// TwinCAT 3 PLC project Contol
// ProgramVersion: 3.1.4023.0
// libraries:
//   Tc2_MC2, * (Beckhoff Automation GmbH)
//   Tc2_MC2_Camming, * (Beckhoff Automation GmbH)
//   Tc2_Standard, * (Beckhoff Automation GmbH)
//   Tc2_System, * (Beckhoff Automation GmbH)
//   Tc2_Utilities, * (Beckhoff Automation GmbH)
//   Tc3_Module, * (Beckhoff Automation GmbH)
//   VisuSymbols,3.5.10.0,System
// project tree:
//   / GlobalTextList.TcGTLO, PlcTask.TcTTO, Visualization Manager.TcVMO (not stored)
//   GVLs/ GVL_UserParamerts.TcGVL
//   POUs/ FB_CsvRead_CamTable.TcPOU, MAIN.TcPOU
//   VISUs/ Visualization.TcVIS
// real-time tasks:
//   TASK PlcTask: cycle T#10ms, priority 20, ADS port 350
// motion (NC):
//   TASK NC-Task 1 SAF: cycle T#2ms, priority 4, ADS port 501
//   TASK NC-Task 1 SVB: cycle T#10ms, priority 8, ADS port 511
//   AXIS master (id 1)
//     OtherSettings: AllowMotionCmdToSlave=true
//     encoder EncType=1
//     drive DrvType=5
//       Analog: TorqueSetpointScale=10, ScaleFactorActTorque=0.1
//       TimeComp: TaskDelayCycles=1
//     controller CtrType=1
//       CtrPara: PriorControlFactor=1
//         Observer: BandWidth=20
//   AXIS Axis 1 (id 2)
//     OtherSettings: AllowMotionCmdToSlave=true
//     encoder EncType=1
//     drive DrvType=5
//       Analog: TorqueSetpointScale=10, ScaleFactorActTorque=0.1
//       TimeComp: TaskDelayCycles=1
//     controller CtrType=1
//       CtrPara: PriorControlFactor=1
//         Observer: BandWidth=20
//   AXIS Axis 2 (id 3)
//     OtherSettings: AllowMotionCmdToSlave=true
//     encoder EncType=1
//     drive DrvType=5
//       Analog: TorqueSetpointScale=10, ScaleFactorActTorque=0.1
//       TimeComp: TaskDelayCycles=1
//     controller CtrType=1
//       CtrPara: PriorControlFactor=1
//         Observer: BandWidth=20
//   AXIS Axis 3 (id 4)
//     OtherSettings: AllowMotionCmdToSlave=true
//     encoder EncType=1
//     drive DrvType=5
//       Analog: TorqueSetpointScale=10, ScaleFactorActTorque=0.1
//       TimeComp: TaskDelayCycles=1
//     controller CtrType=1
//       CtrPara: PriorControlFactor=1
//         Observer: BandWidth=20
//   AXIS Axis 4 (id 5)
//     OtherSettings: AllowMotionCmdToSlave=true
//     encoder EncType=1
//     drive DrvType=5
//       Analog: TorqueSetpointScale=10, ScaleFactorActTorque=0.1
//       TimeComp: TaskDelayCycles=1
//     controller CtrType=1
//       CtrPara: PriorControlFactor=1
//         Observer: BandWidth=20
//   AXIS Axis 5 (id 6)
//     OtherSettings: AllowMotionCmdToSlave=true
//     encoder EncType=1
//     drive DrvType=5
//       Analog: TorqueSetpointScale=10, ScaleFactorActTorque=0.1
//       TimeComp: TaskDelayCycles=1
//     controller CtrType=1
//       CtrPara: PriorControlFactor=1
//         Observer: BandWidth=20
// variable links:
//   Contol/Contol Instance <-> NC-Task 1 SAF/Axes/Axis 1
//     PlcTask Inputs/MAIN.AxMotor[0].NcToPlc <-> Outputs/ToPlc
//     PlcTask Outputs/MAIN.AxMotor[0].PlcToNc <-> Inputs/FromPlc
//   Contol/Contol Instance <-> NC-Task 1 SAF/Axes/Axis 2
//     PlcTask Inputs/MAIN.AxMotor[1].NcToPlc <-> Outputs/ToPlc
//     PlcTask Outputs/MAIN.AxMotor[1].PlcToNc <-> Inputs/FromPlc
//   Contol/Contol Instance <-> NC-Task 1 SAF/Axes/Axis 3
//     PlcTask Inputs/MAIN.AxMotor[2].NcToPlc <-> Outputs/ToPlc
//     PlcTask Outputs/MAIN.AxMotor[2].PlcToNc <-> Inputs/FromPlc
//   Contol/Contol Instance <-> NC-Task 1 SAF/Axes/Axis 4
//     PlcTask Inputs/MAIN.AxMotor[3].NcToPlc <-> Outputs/ToPlc
//     PlcTask Outputs/MAIN.AxMotor[3].PlcToNc <-> Inputs/FromPlc
//   Contol/Contol Instance <-> NC-Task 1 SAF/Axes/Axis 5
//     PlcTask Inputs/MAIN.AxMotor[4].NcToPlc <-> Outputs/ToPlc
//     PlcTask Outputs/MAIN.AxMotor[4].PlcToNc <-> Inputs/FromPlc
//   Contol/Contol Instance <-> NC-Task 1 SAF/Axes/master
//     PlcTask Inputs/MAIN.AXMaster.NcToPlc <-> Outputs/ToPlc
//     PlcTask Outputs/MAIN.AXMaster.PlcToNc <-> Inputs/FromPlc

CONFIGURATION Contol
    RESOURCE PLC ON TwinCAT3
        TASK PlcTask(INTERVAL := T#10ms, PRIORITY := 20);
        PROGRAM MAIN WITH PlcTask : MAIN;
    END_RESOURCE
END_CONFIGURATION

// ---- GVLs/GVL_UserParamerts.TcGVL
//{attribute 'qualified_only'}
VAR_GLOBAL CONSTANT
	// kinetic parameters
	lrVelocity						: REAL		:= 1000;
	lrAcceleration					: REAL		:= 1000;
	lrDeceleration					: REAL		:= 1000;
	
	// show parameters
	rShowVelocity					: REAL		:= 100;
	rShowAcceleration				: REAL		:= 1000;
	rShowDeceleration				: REAL		:= 1000;
	
	// csv file parameters
	iMaxPoints						: INT		:= 5864;		// Maximum number of frames/rows/required positions 32.000 -> Activate Configuration
	iMotorsNum						: INT		:= 5;			// Fixed
	sFileDir						: STRING	:= 'C:\Users\Amr Awad\Desktop\TC_AxesSimulator\_ShowFiles_\';
	sFileName						: STRING	:= 'gesamt_show.csv';
END_VAR
VAR_GLOBAL PERSISTENT
	aa2lrTable						: ARRAY[0..iMotorsNum-1] OF ARRAY[0..iMaxPoints-1,0..1] OF LREAL;
END_VAR

// ---- POUs/MAIN.TcPOU
PROGRAM MAIN
VAR
	fbTimeout						: TON;
	
	(* GUI Parameters *)
	// User Control
	boShowLoad						: BOOL;
	boShowStart						: BOOL;
	boShowPause						: BOOL;
	boShowStop						: BOOL;
	
	(* Show Functions & Parameters *)
	// 1. csv file loading
	fbCsvRead						: FB_CsvRead_CamTable;
	iFrames							: INT;
	boShowLoadError					: BOOL;
	boShowLoading					: BOOL;
	boShowLoaded					: BOOL;
	i								: INT;
	iTable							: INT	:= 0;
	
	// 2. show manupulation
	iShowState						: INT := 0;
	
	// camming table
	TableCamRef						: ARRAY[0..iMotorsNum-1] OF MC_CAM_REF;
	MC_CamTableSelect				: MC_CamTableSelect;
	MC_ReadCamTableCharacteristics	: ARRAY[0..iMotorsNum-1] OF MC_ReadCamTableCharacteristics;
	MC_TableCharacValues			: ARRAY[0..iMotorsNum-1] OF MC_TableCharacValues;
	
	// 1. Master Axis
	AXMaster						: AXIS_REF;
	fbMasterEnable					: MC_Power;
	fbMasterSetPosition				: MC_SetPosition;
	fbMasterMoveAbs					: MC_MoveAbsolute;
	fbMasterStop					: MC_Stop;
	fbMasterReset					: MC_Reset;
	
	boMasterEnable					: BOOL;
	boMasterSetPosition				: BOOL;
	boMasterMovAbs					: BOOL;
	rMasterTargetPosition			: REAL;
	boMasterStop					: BOOL;
	boShowPauseLatch				: BOOL;
	boShowStopLatch					: BOOL;
	boMasterReset					: BOOL;
	
	// 2. Slave Axes
	AxMotor							: ARRAY[0..iMotorsNum-1] OF AXIS_REF;
	fbEnable						: ARRAY[0..iMotorsNum-1] OF MC_Power;
	fbMoveAbs						: ARRAY[0..iMotorsNum-1] OF MC_MoveAbsolute;
	ST_CamInOptions					: ST_CamInOptions;	// Data Type deceleration — MC_CamIn input
	fbCamIn							: ARRAY[0..iMotorsNum-1] OF MC_CamIn;
	fbCamOut						: ARRAY[0..iMotorsNum-1] OF MC_CamOut;
	fbReset							: ARRAY[0..iMotorsNum-1] OF MC_Reset;
	
	boEnable						: BOOL;
	boEnabled						: BOOL;
	boMoveAbs						: BOOL;
	boMoveAbsDone					: BOOL;
	boMoveAbsError					: BOOL;
	boAxCamIn						: BOOL	:= FALSE;
	boAxCamInDone					: BOOL;
	boAxCamOut						: BOOL	:= FALSE;
	boAxCamOutDone					: BOOL;
	boReset							: BOOL;
	
	boShowActived					: BOOL;
END_VAR

// General
boShowLoading										:= fbCsvRead.OUT_boBusy;
boShowLoaded										:= aa2lrTable[iMotorsNum-1][iMaxPoints-1,0] <> 0 AND NOT fbCsvRead.OUT_boBusy;

fbTimeout();

// Logic Control
IF NOT boShowActived THEN
	fbCsvRead(
		IN_smaxDirectoryName		 				:= sFileDir, 
		IN_sFileName								:= sFileName, 
		IN_sColumnSeparator							:= ',', 
		IN_iMotorsNr								:= iMotorsNum, 
		IN_boStartReading							:= boShowLoad, 
		IN_paa2lrTable								:= ADR(aa2lrTable), 
		OUT_boError									=> boShowLoadError);
	IF fbCsvRead.OUT_boDone AND NOT fbCsvRead.OUT_boError THEN
		iFrames										:= fbCsvRead.OUT_iRowsnNumber;
		boShowLoad									:= FALSE;
	ELSIF fbCsvRead.OUT_boDone AND fbCsvRead.OUT_boError THEN
		boShowLoad									:= FALSE;
	END_IF
	IF boShowLoaded AND boShowStart THEN
		boShowActived								:= TRUE;
		iShowState									:= 10;
	END_IF
ELSE
	CASE iShowState OF
		0:		// Idle
			boShowActived							:= FALSE;
			boShowPauseLatch						:= FALSE;
			boShowStopLatch							:= FALSE;
			
		10:		// preparing camming referencing
			rMasterTargetPosition					:= LREAL_TO_REAL(aa2lrTable[0][iMaxPoints-1,0]);	// last time stamp in the table
			FOR i := 0 TO iMotorsNum - 1 DO
				TableCamRef[i].pArray				:= ADR(aa2lrTable[i]);
				TableCamRef[i].ArraySize			:= SIZEOF(aa2lrTable[i]);
				TableCamRef[i].TableType			:= MC_TABLETYPE_NONEQUIDISTANT;
				TableCamRef[i].NoOfRows				:= INT_TO_UDINT(iMaxPoints);
				TableCamRef[i].NoOfColumns			:= 2;
			END_FOR
			iShowState								:= 20;
			
		20:		// select camming table
			MC_CamTableSelect(
				Master								:= AxMaster, 
				Slave								:= AxMotor[iTable], 
				CamTable							:= TableCamRef[iTable], 
				Execute								:= TRUE, 
				Periodic							:= FALSE, 
				MasterAbsolute						:= TRUE, 
				SlaveAbsolute						:= TRUE, 
				CamTableID							:= INT_TO_UDINT(iTable+1), 
				Done=> , 
				Busy=> , 
				Error=> , 
				ErrorID=> );
			IF MC_CamTableSelect.Done AND NOT MC_CamTableSelect.Error THEN
				iTable								:= iTable + 1;
				MC_CamTableSelect(	
					Master							:= AxMaster, 
					Slave							:= AxMotor[iTable], 
					CamTable						:= TableCamRef[iTable],
					Execute							:= FALSE);
				IF iTable = iMotorsNum-1 THEN
					iTable							:= 0;
					iShowState						:= 30;
				ELSE
					//
				END_IF
			ELSIF MC_CamTableSelect.Error THEN
				MC_CamTableSelect(	
					Master							:= AxMaster, 
					Slave							:= AxMotor[iTable], 
					CamTable						:= TableCamRef[iTable],
					Execute							:= FALSE);
				iTable								:= 0;
			END_IF
			
		30:		// kinetic initialization
			fbTimeout.IN							:= TRUE;
			fbTimeout.PT							:= T#5S;
			boMasterEnable							:= TRUE;
			boEnable								:= TRUE;
			boEnabled								:= AXMaster.NcToPlc.StateDWord.0;
			FOR i := 0 TO iMotorsNum - 1 DO
				boEnabled							:= boEnabled AND AxMotor[i].NcToPlc.StateDWord.0;
			END_FOR
			IF boEnabled THEN
				fbTimeout.IN						:= FALSE;
				iShowState							:= 40;
			ELSIF fbTimeout.Q THEN
				fbTimeout.IN						:= FALSE;
				// Error
			END_IF
			
		40:		// Master position reset
			boMasterSetPosition						:= TRUE;
			IF fbMasterSetPosition.Done THEN
				boMasterSetPosition					:= FALSE;
				iShowState							:= 50;
			ELSIF fbMasterSetPosition.Error THEN
				boMasterSetPosition					:= FALSE;
				// Error
			END_IF
			
		50:		// move all axes to the home position
			fbTimeout.IN							:= TRUE;
			fbTimeout.PT							:= T#5S;
			boMoveAbs								:= TRUE;
			boMoveAbsDone							:= TRUE;
			boMoveAbsError							:= FALSE;
			FOR i := 0 TO iMotorsNum - 1 DO
				boMoveAbsDone						:= boMoveAbsDone AND fbMoveAbs[i].Done;
				boMoveAbsError						:= boMoveAbsError OR fbMoveAbs[i].Error;
			END_FOR
			IF boMoveAbsDone AND NOT boMoveAbsError THEN
				fbTimeout.IN						:= FALSE;
				boMoveAbs							:= FALSE;
				iShowState							:= 60;
			ELSIF boMoveAbsError THEN
				fbTimeout.IN						:= FALSE;
				boMoveAbs							:= FALSE;
				// Error
			ELSIF fbTimeout.Q THEN
				fbTimeout.IN						:= FALSE;
				// Error
			END_IF
			
		60:		// couple axes
			fbTimeout.IN							:= TRUE;
			fbTimeout.PT							:= T#5S;
			boAxCamIn								:= TRUE;
			boAxCamInDone							:= TRUE;
			FOR i := 0 TO iMotorsNum - 1 DO
				boAxCamInDone						:= boAxCamInDone AND fbCamIn[i].InSync AND NOT fbCamIn[i].Error;
				IF fbCamIn[i].Error THEN
					// Error
				END_IF
			END_FOR
			IF boAxCamInDone THEN
				fbTimeout.IN						:= FALSE;
				boAxCamIn							:= FALSE;
				iShowState							:= 70;
			ELSIF fbTimeout.Q THEN
				fbTimeout.IN						:= FALSE;
				// Error
			END_IF
			
		70:		// move master axis
			boMasterMovAbs							:= TRUE;
			IF fbMasterMoveAbs.Busy THEN
				boMasterMovAbs						:= FALSE;
				iShowState							:= 75;
			END_IF
			
		75:		// check show end
			IF fbMasterMoveAbs.Done THEN
				iShowState							:= 80;
			END_IF
			IF boShowPause THEN
				boMasterStop						:= TRUE;
				boShowPauseLatch					:= TRUE;
				iShowState							:= 77;
			ELSIF boShowStop THEN
				boMasterStop						:= TRUE;
				boShowStopLatch						:= TRUE;
				iShowState							:= 77;
			END_IF
			
		77:		// stop check
			boMasterStop							:= FALSE;
			IF fbMasterStop.Done THEN
				iShowState							:= 78;
			END_IF
			
		78:		// decision making
			IF boShowPauseLatch AND boShowStart THEN
				boShowPauseLatch					:= FALSE;
				iShowState							:= 70;
			END_IF
			IF boShowStopLatch THEN
				iShowState							:= 80;
			END_IF
			
		80:		// decouple axes
			fbTimeout.IN							:= TRUE;
			fbTimeout.PT							:= T#5S;
			boAxCamOut								:= TRUE;
			boAxCamOutDone							:= TRUE;
			FOR i := 0 TO iMotorsNum - 1 DO
				boAxCamOutDone						:= boAxCamOutDone AND fbCamOut[i].Done AND NOT fbCamOut[i].Error;
				IF fbCamOut[i].Error THEN
					// Error
				END_IF
			END_FOR
			IF boAxCamOutDone THEN
				fbTimeout.IN						:= FALSE;
				boAxCamOut							:= FAlse;
				IF boShowStopLatch THEN
					boShowStopLatch					:= FALSE;
					iShowState						:= 0;
				ELSE
					iShowState						:= 40;
				END_IF
			ELSIF fbTimeout.Q THEN
				fbTimeout.IN						:= FALSE;
				// Error
			END_IF
	END_CASE
END_IF

(* Cyclic Calls *)
// 1. Master Axis
fbMasterEnable(
	Axis											:= AxMaster, 
	Enable											:= boMasterEnable, 
	Enable_Positive									:= TRUE, 
	Enable_Negative									:= TRUE, 
	Override										:= 100, 
	BufferMode										:= MC_Aborting, 
	Options:= , 
	Status=> , 
	Busy=> , 
	Active=> , 
	Error=> , 
	ErrorID=> );

fbMasterSetPosition(
	Axis											:= AxMaster, 
	Execute											:= boMasterSetPosition, 
	Position										:= 0, 
	Mode:= , 
	Options:= , 
	Done=> , 
	Busy=> , 
	Error=> , 
	ErrorID=> );

fbMasterMoveAbs(
	Axis											:= AxMaster, 
	Execute											:= boMasterMovAbs, 
	Position										:= rMasterTargetPosition, 
	Velocity										:= rShowVelocity, 
	Acceleration									:= rShowAcceleration, 
	Deceleration									:= rShowDeceleration, 
	Jerk:= , 
	BufferMode:= , 
	Options:= , 
	Done=> , 
	Busy=> , 
	Active=> , 
	CommandAborted=> , 
	Error=> , 
	ErrorID=> );

fbMasterStop(
	Axis											:= AxMaster, 
	Execute											:= boMasterStop, 
	Deceleration:= , 
	Jerk:= , 
	Options:= , 
	Done=> , 
	Busy=> , 
	Active=> , 
	CommandAborted=> , 
	Error=> , 
	ErrorID=> );

fbMasterReset(
	Axis											:= AxMaster, 
	Execute											:= boMasterReset, 
	Done=> , 
	Busy=> , 
	Error=> , 
	ErrorID=> );

// 2. Pendulum Axis
FOR i := 0 TO iMotorsNum-1 DO
	fbEnable[i](
		Axis										:= AxMotor[i], 
		Enable										:= boEnable, 
		Enable_Positive								:= TRUE, 
		Enable_Negative								:= TRUE, 
		Override:= , 
		BufferMode:= , 
		Options:= , 
		Status=> , 
		Busy=> , 
		Active=> , 
		Error=> , 
		ErrorID=> );
	
	fbMoveAbs[i](
		Axis										:= AxMotor[i], 
		Execute										:= boMoveAbs, 
		Position									:= aa2lrTable[i][0, 1], 
		Velocity									:= lrVelocity, 
		Acceleration								:= lrAcceleration, 
		Deceleration								:= lrDeceleration, 
		Jerk:= , 
		BufferMode:= , 
		Options:= , 
		Done=> , 
		Busy=> , 
		Active=> , 
		CommandAborted=> , 
		Error=> , 
		ErrorID=> );
	
	fbCamIn[i](
		Master										:= AxMaster, 
		Slave										:= AxMotor[i], 
		Execute										:= boAxCamIn, 
		MasterOffset								:= 0, 
		SlaveOffset									:= 0, 
		MasterScaling								:= 1, 
		SlaveScaling								:= 1, 
		StartMode:= , 
		CamTableID									:= 1, 
		BufferMode:= , 
		Options										:= ST_CamInOptions, 
		//InterpolationType							:= MC_InterpolationType_Spline, 
		InSync=> , 
		Busy=> , 
		Active=> , 
		CommandAborted=> , 
		Error=> , 
		ErrorID=> );
	
	fbCamOut[i](
		Slave										:= AxMotor[i], 
		Execute										:= boAxCamOut, 
		Options:= , 
		Done=> , 
		Busy=> , 
		Error=> , 
		ErrorID=> );
	
	fbReset[i](
		Axis										:= AxMotor[i], 
		Execute										:= boReset, 
		Done=> , 
		Busy=> , 
		Error=> , 
		ErrorID=> );
END_FOR

END_PROGRAM

// ---- POUs/FB_CsvRead_CamTable.TcPOU
FUNCTION_BLOCK FB_CsvRead_CamTable
VAR_INPUT
	IN_smaxDirectoryName				: T_MaxString;
	IN_sFileName						: STRING;
	IN_sColumnSeparator					: STRING;
	IN_iMotorsNr						: INT;
	IN_boStartReading					: BOOL;
	IN_paa2lrTable						: POINTER TO ARRAY[0..iMotorsNum-1] OF ARRAY[0..iMaxPoints-1,0..1] OF LREAL;
END_VAR
VAR_OUTPUT
	OUT_boBusy							: BOOL;		// Reading active
	OUT_boDone							: BOOL;		// Reading Done user-defined flag
	OUT_boError							: BOOL;
	OUT_iReadingError					: INT;		// Reading error user-defined flag; 0:Clear, 1:Opening, 2:Getting
	OUT_iRowsnNumber					: INT;		// Number of actual read rows
	//OUT_arTableColumn					: ARRAY[0..iMotorsNum] OF ARRAY[0..iMaxPoints-1] OF REAL;
END_VAR

VAR
	ReadCSV								: R_TRIG;
	iStep								: INT;						// identifier of the execution sequence — State index
	
	fbFileOpen							: FB_FileOpen;				// Opens file
	fbFileGets							: FB_FileGets;				// Reads text data from the opened file
	fbReader							: FB_CSVMemBufferReader;	// Helper function block used to parse CSV data bytes
	fbFileClose							: FB_FileClose;				// Closes file
	
	sPathName							: T_MaxString;
	nMode								: DWORD := FOPEN_MODEREAD OR FOPEN_MODEBINARY;	(* FileOpen input *)
	bBusy								: BOOL;											(* Internal Busy flag *)
	nErrId								: UDINT;										(* Block output *)
	hFile								: UINT	:= 0;									(* File handle of the source file *)
	
	iRow								: INT;											// Row number (record)
	iColumn								: INT;											// Column number (record field)
	
	lrDummy								: LREAL;
END_VAR

ReadCSV(CLK								:= IN_boStartReading);	// Latching the start reading command
OUT_boBusy								:= iStep <> 0;			// Busy as long as state machine running

// Column Separator selection
IF IN_sColumnSeparator = ',' THEN
	DEFAULT_CSV_FIELD_SEP				:= 16#2C;				// American Separator (,) 16#2C
ELSIF IN_sColumnSeparator = ';' THEN
	DEFAULT_CSV_FIELD_SEP				:= 16#3B;				// European Separator (;) 16#3B
END_IF

CASE iStep OF 
	0:		// Sleep Mode — wait till the starting signal is triggered
		sPathName						:= CONCAT(IN_smaxDirectoryName, IN_sFileName);
		fbFileOpen(bExecute				:= FALSE);
		fbFileGets(bExecute				:= FALSE);
		IF ReadCSV.Q THEN	// Reset parameters — Transition to the next step
			OUT_boDone			:= FALSE;
			OUT_iReadingError			:= 0;
			MEMSET(IN_paa2lrTable, 0, SIZEOF(IN_paa2lrTable^));
			bBusy						:= TRUE;
			OUT_boError					:= FALSE;
			nErrId						:= 0;
			hFile						:= 0;
			iRow						:= 0;
			iStep						:= 10;
		END_IF
	
	10:		// File Opening Command
		fbFileOpen(	
			sPathName					:= sPathName, 
			nMode						:= nMode, 
			bExecute					:= TRUE, 
			bError						=> OUT_boError, 
			nErrID 						=> nErrID, 
			hFile						=> hFile );
		IF NOT fbFileOpen.bBusy THEN
			IF NOT fbFileOpen.bError THEN
				fbFileOpen(bExecute		:= FALSE);
				iStep					:= 20;      // File opened & without error
			ELSE
				fbFileOpen(bExecute		:= FALSE);
				iStep					:= 100;    // Error — File not found!
				OUT_iReadingError		:= 1;
			END_IF
		END_IF
		
	20:		// Data Getting Command
		fbFileGets(	
			hFile						:= hFile, 
			bExecute					:= TRUE, 
			bError						=> OUT_boError);
		IF NOT fbFileGets.bBusy THEN
			IF NOT fbFileGets.bError THEN
				IF fbFileGets.bEOF THEN
					fbFileGets(bExecute	:= FALSE);
					iStep				:= 40;		// .csv file end is reached — Close File
				ELSE
					fbFileGets(bExecute	:= FALSE);
					iStep				:= 30;		// Parse text data
				END_IF
			ELSE
				iStep					:= 100;		// Error — During the excution!
				OUT_iReadingError		:= 2;
			END_IF		
		END_IF
		
	30:		// Parse text data
		fbReader(	
			eCmd						:= eEnumCmd_First, 
			pBuffer						:= ADR(fbFileGets.sLine), 
			cbBuffer					:= SIZEOF(fbFileGets.sLine));	// Read first field value — given from the manual
		IF fbReader.bOk THEN
			lrDummy						:= STRING_TO_LREAL(fbReader.getValue);
			FOR iColumn := 0 TO IN_iMotorsNr-1 DO
				fbReader(	
					eCmd				:= eEnumCmd_Next, 
					pBuffer				:= ADR(fbFileGets.sLine), 
					cbBuffer			:= SIZEOF(fbFileGets.sLine));
				IN_paa2lrTable^[iColumn][iRow,0]	:= lrDummy;								// Master Axis Positions
				IN_paa2lrTable^[iColumn][iRow,1]	:= STRING_TO_REAL(fbReader.getValue);	// Motors Axes Positions
			END_FOR
			iRow						:= iRow +1;		// Increment number of read records
			iStep						:= 20;			// Read new row
		END_IF
	
	40:		// Close source file command
		OUT_iRowsnNumber				:= iRow;
		fbFileClose(	
			hFile						:= hFile, 
			bExecute					:= TRUE, 
			bError						=> OUT_boError);
		IF NOT fbFileClose.bBusy THEN
			fbFileClose(bExecute		:= FALSE);
			hFile						:= 0;
			iStep						:= 100;
		END_IF
	
	100:	// Error OR ready step => cleanup
		IF ( hFile <> 0 ) THEN
			iStep						:= 10;		// Close the source file and cleanup hFile
		ELSE
			bBusy						:= FALSE;	// Lowering the Busy flag
			OUT_boDone			:= TRUE;	// Ending Service Routine flag
			iStep						:= 0;		// Ready for a new run when triggered/called
		END_IF
END_CASE

END_FUNCTION_BLOCK

// ---- GlobalTextList.TcGTLO
TEXTLIST GlobalTextList
  628 = 'Axes Coupled'
  409 = 'Control'
  464 = 'Feadback'
  166 = 'Show Activated'
  915 = 'Show Load'
  700 = 'Show Loaded'
  942 = 'Show Loading'
  86 = 'Show Pause'
  299 = 'Show Running'
  447 = 'Show Start'
  735 = 'Show Stop'
END_TEXTLIST

// ---- VISUs/Visualization.TcVIS
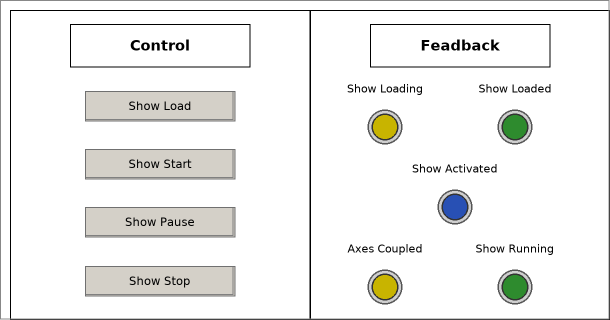
VISUALIZATION Visualization  // 610x320
    Rectangle (310,10 300x310)
    Rectangle (10,10 300x310)
    Button (85,91 150x30), "Show Load", input disabled if: MAIN.boShowActived OR MAIN.fbCsvRead.OUT_boBusy
        tap MAIN.boShowLoad
    Rectangle (70,24 180x43), "Control"
    Button (85,149 150x30), "Show Start", input disabled if: (MAIN.boShowActived AND NOT MAIN.boShowPauseLatch)OR MAIN.fbCsvRead.OUT_boBusy
        tap MAIN.boShowStart
    Button (85,207 150x30), "Show Pause", input disabled if: NOT MAIN.fbMasterMoveAbs.Busy
        tap MAIN.boShowPause
    Button (85,266 150x30), "Show Stop", input disabled if: NOT MAIN.fbMasterMoveAbs.Busy
        tap MAIN.boShowStop
    Rectangle (370,24 180x43), "Feadback"
    Lamp1 (365,107 40x40), variable: MAIN.boShowLoading, style: Lamp-Lamp1-Yellow
    Rectangle (335,79 100x20), "Show Loading"
    Lamp1 (495,107 40x40), variable: MAIN.boShowLoaded, style: Lamp-Lamp1-Green
    Rectangle (465,79 100x20), "Show Loaded"
    Lamp1 (435,187 40x40), variable: MAIN.boShowActived, style: Lamp-Lamp1-Blue
    Rectangle (405,159 100x20), "Show Activated"
    Lamp1 (365,267 40x40), variable: MAIN.AXMaster.NcToPlc.CoupleState = 1, style: Lamp-Lamp1-Yellow
    Rectangle (335,239 100x20), "Axes Coupled"
    Lamp1 (495,267 40x40), variable: MAIN.fbMasterMoveAbs.Busy, style: Lamp-Lamp1-Green
    Rectangle (465,239 100x20), "Show Running"
END_VISUALIZATION
